Universal Robots PolyScope program: poner_en_posicion.urp

Program poner_en_posicion (installation=default directory=/programs createdIn=5.14.5 lastSavedIn=5.14.5 robotSerialNumber=20195300809)
Calibrated DH parameters: a=[-0.000085, -0.20076, -0.212369, 0.000121, -0.000118, 0]; d=[0.15185, -26.306375, 24.753047, 1.684739, 0.085386, 0.092088]; alpha=[1.572149, -0.00522, -0.011864, 1.571339, -1.571085, 0]; deltaTheta=[0, 0.599885, -0.513355, -0.086555, 0.000006, 0]
InitVariablesNode
Robot Program (runOnlyOnce=false)
  MoveJ speed 60 deg/s, acceleration 80 deg/s^2 (useActiveTCP=true) feature=Base
    Waypoint Posicion_foto: TCP in base x=-241.348 y=-154.076 z=452.935 mm, rx=-1.8451 ry=-1.9333 rz=0.6043 rad; joints [6.803, -85.736, 5.234, -43.66, -92.516, 4.131] deg; TCP offset x=0 y=0 z=150 mm, rx=0 ry=0 rz=0 rad
    URCap Gripper Activate (Robotiq_Grippers, Robotiq Inc.) dataModel(ResetAndActivateKey=false)
